FUNCTION_BLOCK MonostableCylinder EXTENDS BaseCylinder
VAR_INPUT
END_VAR
VAR_OUTPUT
END_VAR
VAR
END_VAR

METHOD METH_Extend : BOOL
DO_Extend := TRUE;
END_METHOD

METHOD METH_Retract : BOOL
DO_Extend := FALSE;
END_METHOD

END_FUNCTION_BLOCK

(* stored: Version 1.1.0.1
   POU MonostableCylinder: Id {a18c699b-bd3d-4aeb-ae53-a8277b332972}, SpecialFunc None
   Method METH_Extend: Id {05f5864d-e852-4243-969e-e1503423c54c}
   Method METH_Retract: Id {2d449a69-bcb5-47d6-8e7e-d955df080b59} *)
